// TIA Portal V18 export
FUNCTION "TEMPLATE--v1.0--08_Gate Manager" : Void   // FC25, F_LAD
TITLE = Manage Safety Doors
{ S7_Optimized_Access := 'TRUE' }
// v1.0 First Emission
   VAR_TEMP
      temp_EXAMPLE_OPEN : Bool;
   END_VAR
BEGIN

REGION Network 1: Transfer Data from Speed Control
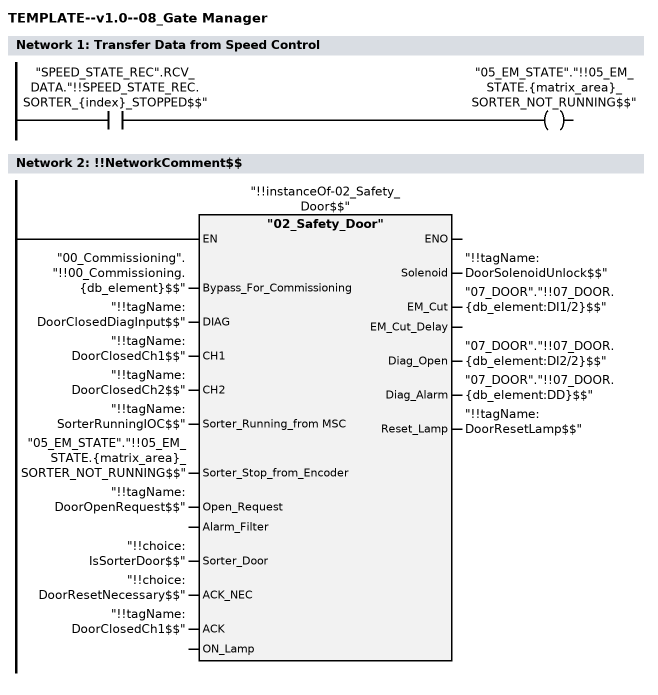
   RUNG wire#powerrail
      Contact( "SPEED_STATE_REC".RCV_DATA."!!SPEED_STATE_REC.SORTER_{index}_STOPPED$$" )
      Coil( "05_EM_STATE"."!!05_EM_STATE.{matrix_area}_SORTER_NOT_RUNNING$$" )
   END_RUNG
   // the same network as SCL:
   "05_EM_STATE"."!!05_EM_STATE.{matrix_area}_SORTER_NOT_RUNNING$$" := "SPEED_STATE_REC".RCV_DATA."!!SPEED_STATE_REC.SORTER_{index}_STOPPED$$";
END_REGION

REGION Network 2: !!NetworkComment$$
   RUNG wire#powerrail
      "!!instanceOf-02_Safety_Door$$"(Bypass_For_Commissioning := "00_Commissioning"."!!00_Commissioning.{db_element}$$", DIAG := "!!tagName:DoorClosedDiagInput$$", CH1 := "!!tagName:DoorClosedCh1$$", CH2 := "!!tagName:DoorClosedCh2$$", "Sorter_Running_from MSC" := "!!tagName:SorterRunningIOC$$", Sorter_Stop_from_Encoder := "05_EM_STATE"."!!05_EM_STATE.{matrix_area}_SORTER_NOT_RUNNING$$", Open_Request := "!!tagName:DoorOpenRequest$$", Alarm_Filter :=, Sorter_Door := "!!choice:IsSorterDoor$$", ACK_NEC := "!!choice:DoorResetNecessary$$", ACK := "!!tagName:DoorClosedCh1$$", ON_Lamp :=, Solenoid => "!!tagName:DoorSolenoidUnlock$$", EM_Cut => "07_DOOR"."!!07_DOOR.{db_element:DI1/2}$$", EM_Cut_Delay =>, Diag_Open => "07_DOOR"."!!07_DOOR.{db_element:DI2/2}$$", Diag_Alarm => "07_DOOR"."!!07_DOOR.{db_element:DD}$$", Reset_Lamp => "!!tagName:DoorResetLamp$$")
   END_RUNG
   // the same network as SCL:
   "!!instanceOf-02_Safety_Door$$"(Bypass_For_Commissioning := "00_Commissioning"."!!00_Commissioning.{db_element}$$",   // "02_Safety_Door"
                           DIAG := "!!tagName:DoorClosedDiagInput$$",
                           CH1 := "!!tagName:DoorClosedCh1$$",
                           CH2 := "!!tagName:DoorClosedCh2$$",
                           "Sorter_Running_from MSC" := "!!tagName:SorterRunningIOC$$",
                           Sorter_Stop_from_Encoder := "05_EM_STATE"."!!05_EM_STATE.{matrix_area}_SORTER_NOT_RUNNING$$",
                           Open_Request := "!!tagName:DoorOpenRequest$$",
                           Sorter_Door := "!!choice:IsSorterDoor$$",
                           ACK_NEC := "!!choice:DoorResetNecessary$$",
                           ACK := "!!tagName:DoorClosedCh1$$",
                           Solenoid => "!!tagName:DoorSolenoidUnlock$$",
                           EM_Cut => "07_DOOR"."!!07_DOOR.{db_element:DI1/2}$$",
                           Diag_Open => "07_DOOR"."!!07_DOOR.{db_element:DI2/2}$$",
                           Diag_Alarm => "07_DOOR"."!!07_DOOR.{db_element:DD}$$",
                           Reset_Lamp => "!!tagName:DoorResetLamp$$");
END_REGION
END_FUNCTION
